(* Logix 5000 project; controller cal1632 1756-L62 rev 16.20; software revision 16.05; part 8 of 57 *)
(* tags used below, declared in another part *)
   FAULT : BOOL;
   p01_r15_footage_ft : REAL;
   p01_real_to_hmi : REAL[112];
   p01r09_pb_global_reset : BOOL;
   p02_real_to_hmi : hmi_real;
   p02r06 : routine;
   p02r06_timer_fault : TIMER[4];
   p02r06_timer_warning : TIMER[4];
   p02r07 : routine;
   p02r07_timer_fault : TIMER[4];
   p02r07_timer_warning : TIMER[4];
   p02r08 : routine;
   p02r08_timer_fault : TIMER[4];
   p02r08_timer_warning : TIMER[4];
   p02r09 : routine;
   p02r09_timer_fault : TIMER[4];
   p02r09_timer_warning : TIMER[4];
   p02r10 : routine;
   p02r10_timer_fault : TIMER[4];
   p02r10_timer_warning : TIMER[4];
   p02r11 : routine;
   p02r11_timer_fault : TIMER[4];
   p02r11_timer_warning : TIMER[4];
   p11_real_to_hmi : REAL[112];
   p12_real_to_hmi : REAL[112];
   p13_real_to_hmi : REAL[112];
   p19_real_to_hmi : REAL[80];
   p20_real_to_hmi : REAL[112];
   p21_real_to_hmi : REAL[112];
   p22_real_to_hmi : REAL[112];
   p23_real_to_hmi : REAL[112];
   p24_real_to_hmi : REAL[112];
   p25_real_to_hmi : REAL[112];
   p26_real_to_hmi : REAL[112];
   p27_real_to_hmi : REAL[112];
   p28_real_to_hmi : REAL[112];
   p29_real_to_hmi : REAL[112];
(* P02_MOP_HMI_Iface, continued *)

ROUTINE R06_Real_to_HMI   (* ladder *)
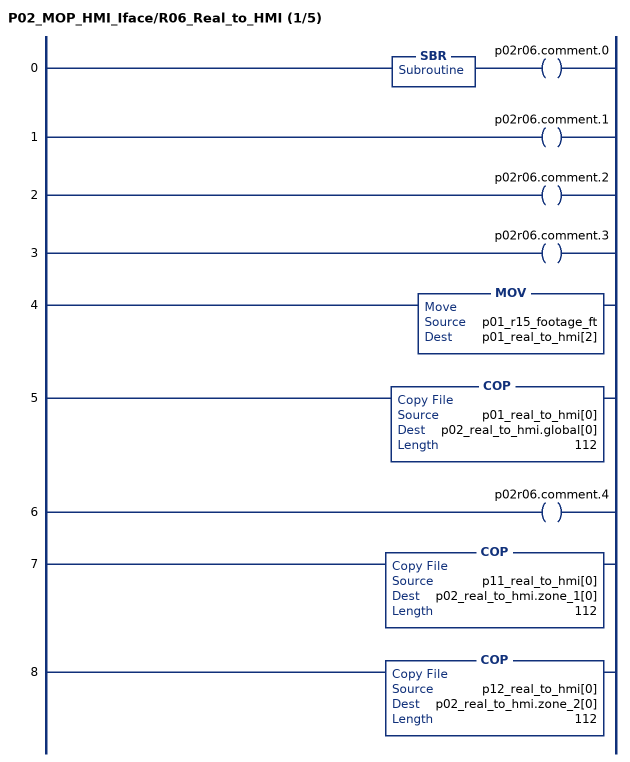
   0: SBR()OTE(p02r06.comment.0);
   1: OTE(p02r06.comment.1);
   2: OTE(p02r06.comment.2);
   3: OTE(p02r06.comment.3);
   4: MOV(p01_r15_footage_ft,p01_real_to_hmi[2]);
   5: COP(p01_real_to_hmi[0],p02_real_to_hmi.global[0],112);
   6: OTE(p02r06.comment.4);
   7: COP(p11_real_to_hmi[0],p02_real_to_hmi.zone_1[0],112);
   8: COP(p12_real_to_hmi[0],p02_real_to_hmi.zone_2[0],112);
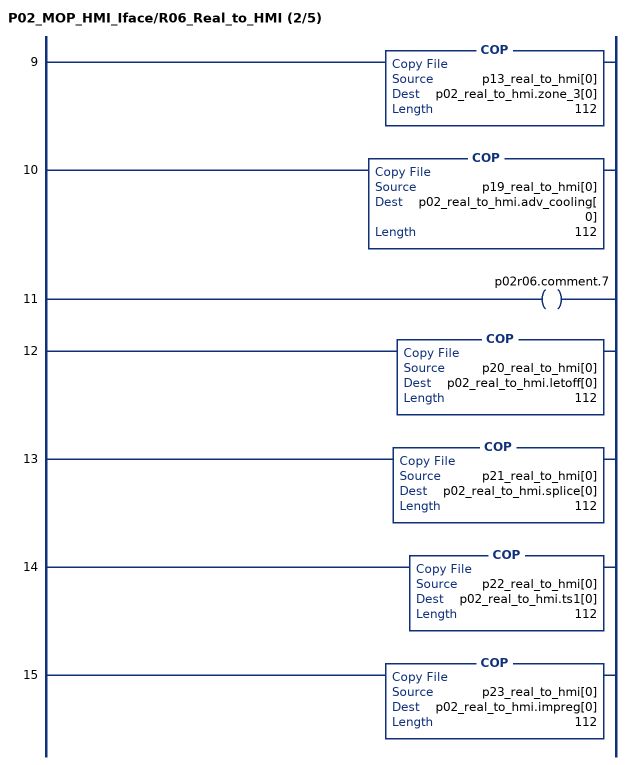
   9: COP(p13_real_to_hmi[0],p02_real_to_hmi.zone_3[0],112);
   10: COP(p19_real_to_hmi[0],p02_real_to_hmi.adv_cooling[0],112);
   11: OTE(p02r06.comment.7);
   12: COP(p20_real_to_hmi[0],p02_real_to_hmi.letoff[0],112);
   13: COP(p21_real_to_hmi[0],p02_real_to_hmi.splice[0],112);
   14: COP(p22_real_to_hmi[0],p02_real_to_hmi.ts1[0],112);
   15: COP(p23_real_to_hmi[0],p02_real_to_hmi.impreg[0],112);
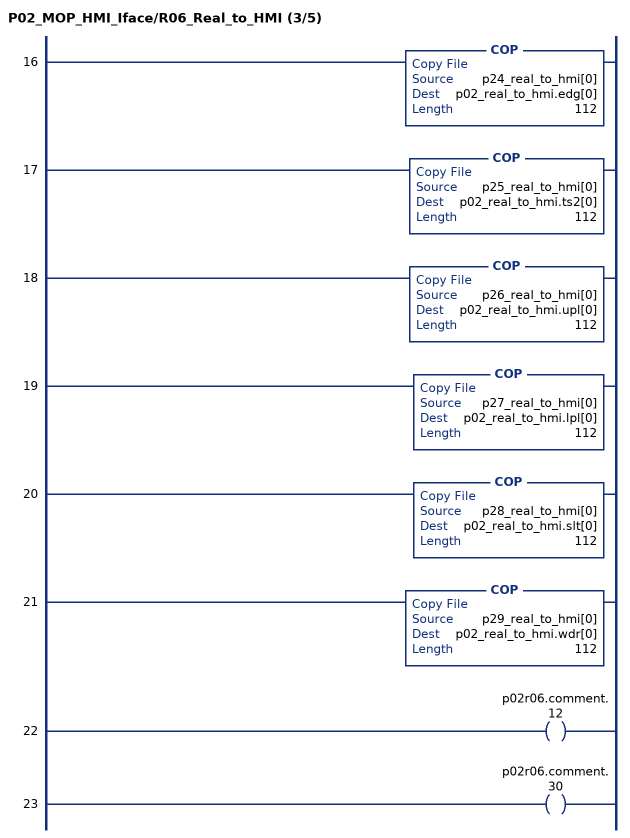
   16: COP(p24_real_to_hmi[0],p02_real_to_hmi.edg[0],112);
   17: COP(p25_real_to_hmi[0],p02_real_to_hmi.ts2[0],112);
   18: COP(p26_real_to_hmi[0],p02_real_to_hmi.upl[0],112);
   19: COP(p27_real_to_hmi[0],p02_real_to_hmi.lpl[0],112);
   20: COP(p28_real_to_hmi[0],p02_real_to_hmi.slt[0],112);
   21: COP(p29_real_to_hmi[0],p02_real_to_hmi.wdr[0],112);
   22: OTE(p02r06.comment.12);
   23: OTE(p02r06.comment.30);
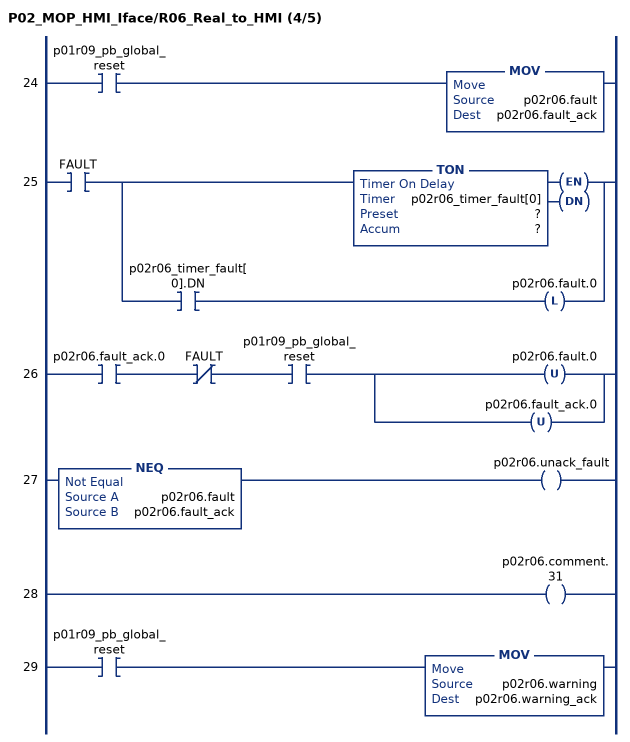
   24: XIC(p01r09_pb_global_reset)MOV(p02r06.fault,p02r06.fault_ack);
   25: XIC(FAULT)[TON(p02r06_timer_fault[0],?,?) ,XIC(p02r06_timer_fault[0].DN) OTL(p02r06.fault.0) ];
   26: XIC(p02r06.fault_ack.0)XIO(FAULT)XIC(p01r09_pb_global_reset)[OTU(p02r06.fault.0) ,OTU(p02r06.fault_ack.0) ];
   27: NEQ(p02r06.fault,p02r06.fault_ack)OTE(p02r06.unack_fault);
   28: OTE(p02r06.comment.31);
   29: XIC(p01r09_pb_global_reset)MOV(p02r06.warning,p02r06.warning_ack);
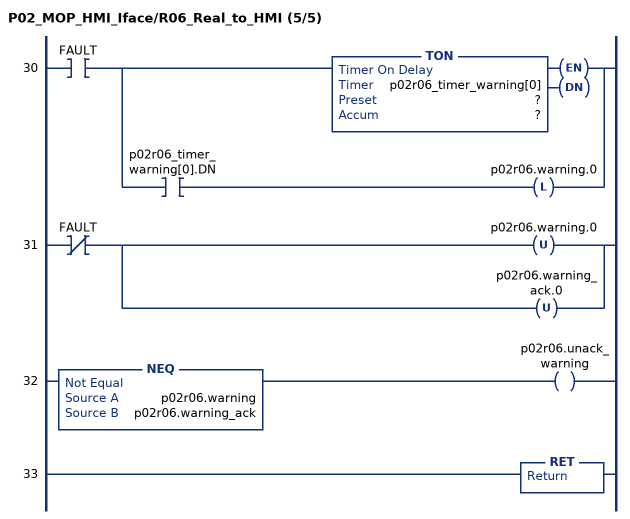
   30: XIC(FAULT)[TON(p02r06_timer_warning[0],?,?) ,XIC(p02r06_timer_warning[0].DN) OTL(p02r06.warning.0) ];
   31: XIO(FAULT)[OTU(p02r06.warning.0) ,OTU(p02r06.warning_ack.0) ];
   32: NEQ(p02r06.warning,p02r06.warning_ack)OTE(p02r06.unack_warning);
   33: RET();
END_ROUTINE

ROUTINE R07_Alarms   (* ladder *)
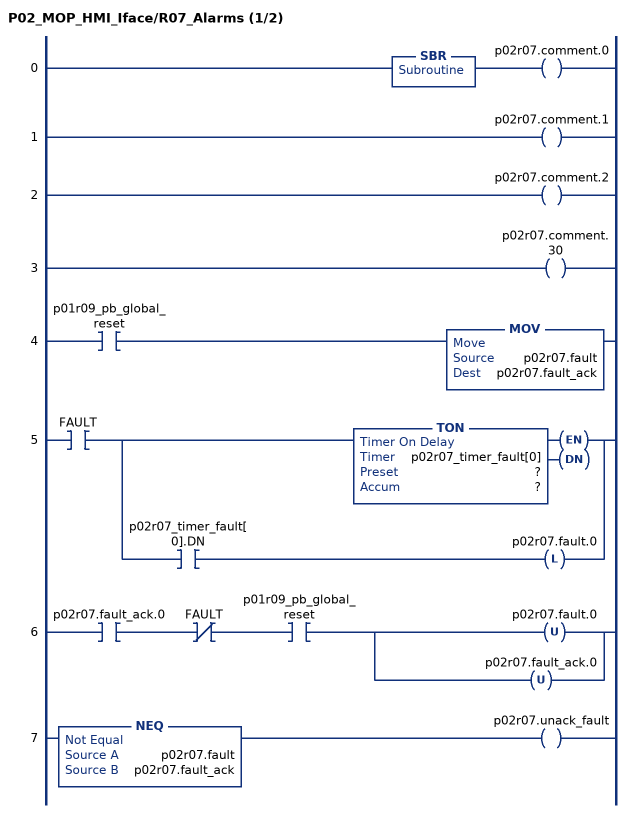
   0: SBR()OTE(p02r07.comment.0);
   1: OTE(p02r07.comment.1);
   2: OTE(p02r07.comment.2);
   3: OTE(p02r07.comment.30);
   4: XIC(p01r09_pb_global_reset)MOV(p02r07.fault,p02r07.fault_ack);
   5: XIC(FAULT)[TON(p02r07_timer_fault[0],?,?) ,XIC(p02r07_timer_fault[0].DN) OTL(p02r07.fault.0) ];
   6: XIC(p02r07.fault_ack.0)XIO(FAULT)XIC(p01r09_pb_global_reset)[OTU(p02r07.fault.0) ,OTU(p02r07.fault_ack.0) ];
   7: NEQ(p02r07.fault,p02r07.fault_ack)OTE(p02r07.unack_fault);
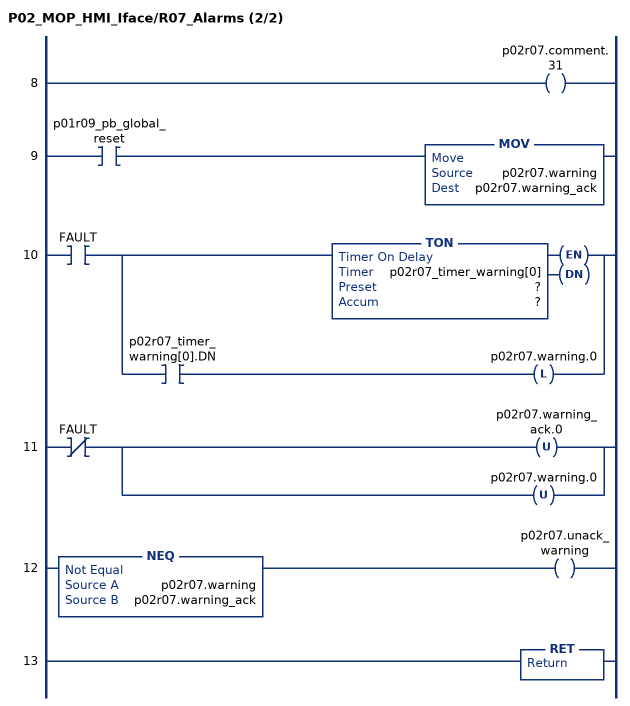
   8: OTE(p02r07.comment.31);
   9: XIC(p01r09_pb_global_reset)MOV(p02r07.warning,p02r07.warning_ack);
   10: XIC(FAULT)[TON(p02r07_timer_warning[0],?,?) ,XIC(p02r07_timer_warning[0].DN) OTL(p02r07.warning.0) ];
   11: XIO(FAULT)[OTU(p02r07.warning_ack.0) ,OTU(p02r07.warning.0) ];
   12: NEQ(p02r07.warning,p02r07.warning_ack)OTE(p02r07.unack_warning);
   13: RET();
END_ROUTINE

ROUTINE R08_Warnings   (* ladder *)
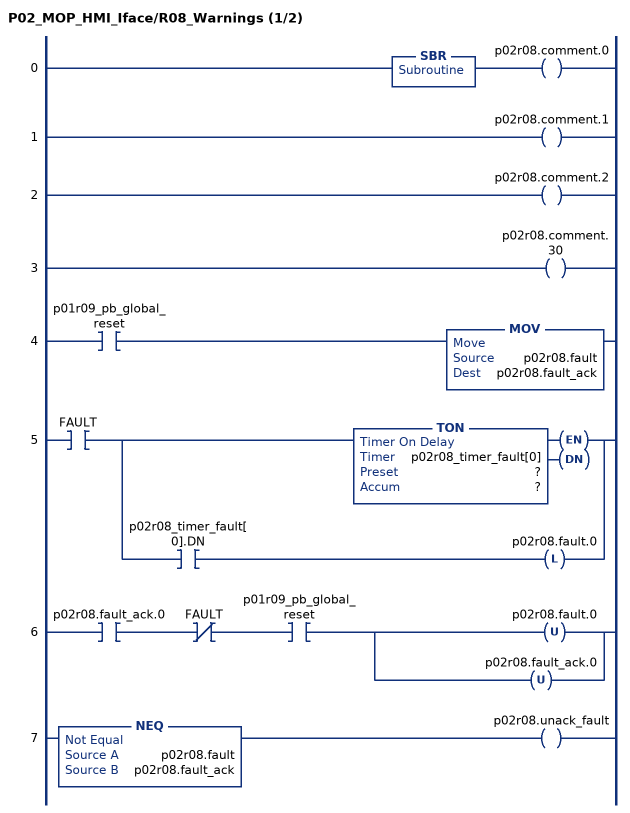
   0: SBR()OTE(p02r08.comment.0);
   1: OTE(p02r08.comment.1);
   2: OTE(p02r08.comment.2);
   3: OTE(p02r08.comment.30);
   4: XIC(p01r09_pb_global_reset)MOV(p02r08.fault,p02r08.fault_ack);
   5: XIC(FAULT)[TON(p02r08_timer_fault[0],?,?) ,XIC(p02r08_timer_fault[0].DN) OTL(p02r08.fault.0) ];
   6: XIC(p02r08.fault_ack.0)XIO(FAULT)XIC(p01r09_pb_global_reset)[OTU(p02r08.fault.0) ,OTU(p02r08.fault_ack.0) ];
   7: NEQ(p02r08.fault,p02r08.fault_ack)OTE(p02r08.unack_fault);
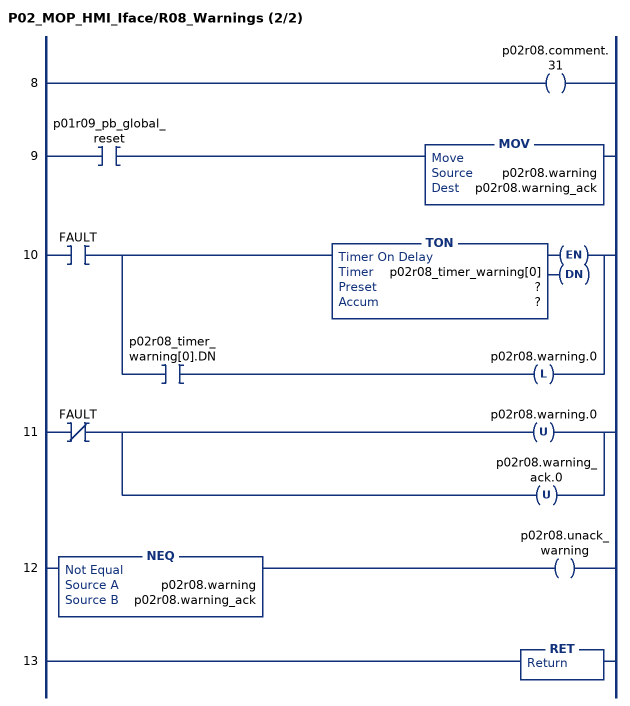
   8: OTE(p02r08.comment.31);
   9: XIC(p01r09_pb_global_reset)MOV(p02r08.warning,p02r08.warning_ack);
   10: XIC(FAULT)[TON(p02r08_timer_warning[0],?,?) ,XIC(p02r08_timer_warning[0].DN) OTL(p02r08.warning.0) ];
   11: XIO(FAULT)[OTU(p02r08.warning.0) ,OTU(p02r08.warning_ack.0) ];
   12: NEQ(p02r08.warning,p02r08.warning_ack)OTE(p02r08.unack_warning);
   13: RET();
END_ROUTINE

ROUTINE R09_Maintenance   (* ladder *)
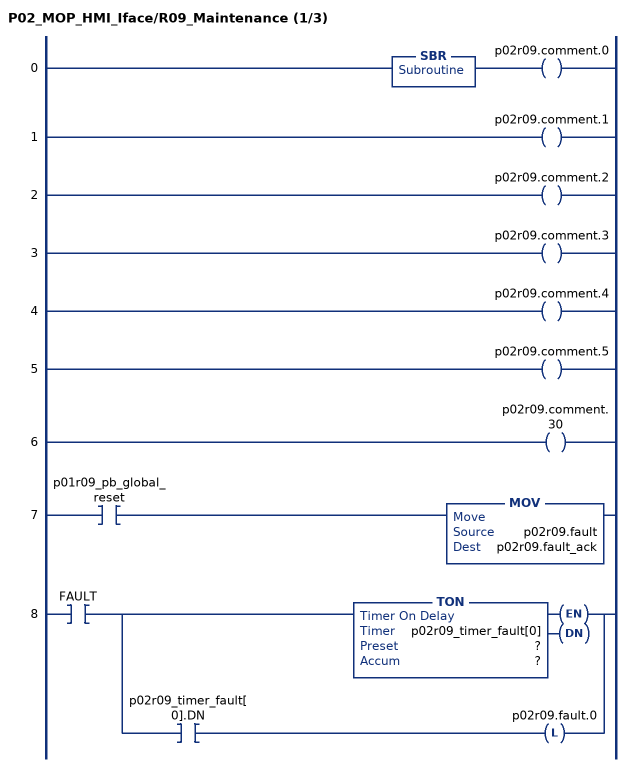
   0: SBR()OTE(p02r09.comment.0);
   1: OTE(p02r09.comment.1);
   2: OTE(p02r09.comment.2);
   3: OTE(p02r09.comment.3);
   4: OTE(p02r09.comment.4);
   5: OTE(p02r09.comment.5);
   6: OTE(p02r09.comment.30);
   7: XIC(p01r09_pb_global_reset)MOV(p02r09.fault,p02r09.fault_ack);
   8: XIC(FAULT)[TON(p02r09_timer_fault[0],?,?) ,XIC(p02r09_timer_fault[0].DN) OTL(p02r09.fault.0) ];
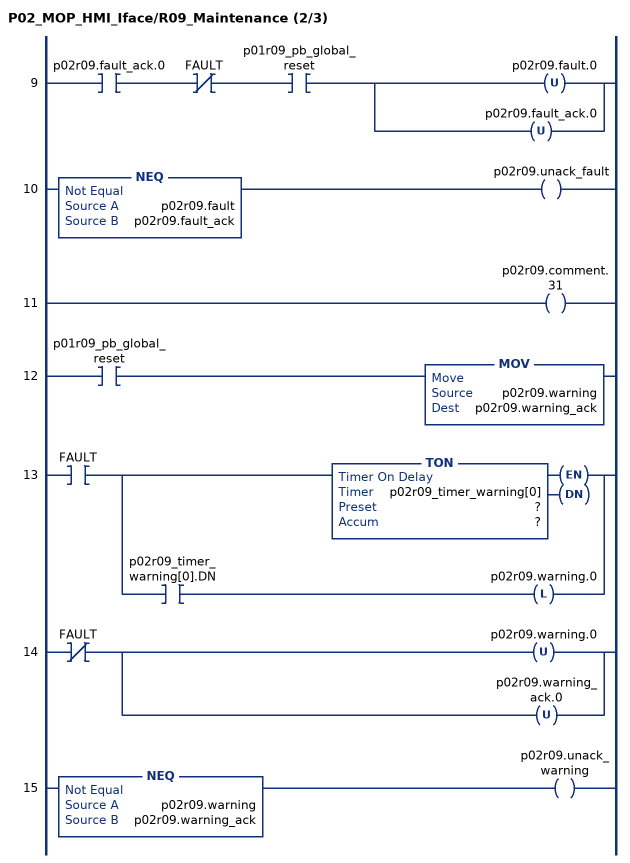
   9: XIC(p02r09.fault_ack.0)XIO(FAULT)XIC(p01r09_pb_global_reset)[OTU(p02r09.fault.0) ,OTU(p02r09.fault_ack.0) ];
   10: NEQ(p02r09.fault,p02r09.fault_ack)OTE(p02r09.unack_fault);
   11: OTE(p02r09.comment.31);
   12: XIC(p01r09_pb_global_reset)MOV(p02r09.warning,p02r09.warning_ack);
   13: XIC(FAULT)[TON(p02r09_timer_warning[0],?,?) ,XIC(p02r09_timer_warning[0].DN) OTL(p02r09.warning.0) ];
   14: XIO(FAULT)[OTU(p02r09.warning.0) ,OTU(p02r09.warning_ack.0) ];
   15: NEQ(p02r09.warning,p02r09.warning_ack)OTE(p02r09.unack_warning);
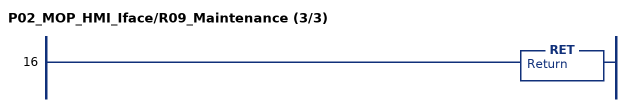
   16: RET();
END_ROUTINE

ROUTINE R10   (* ladder *)
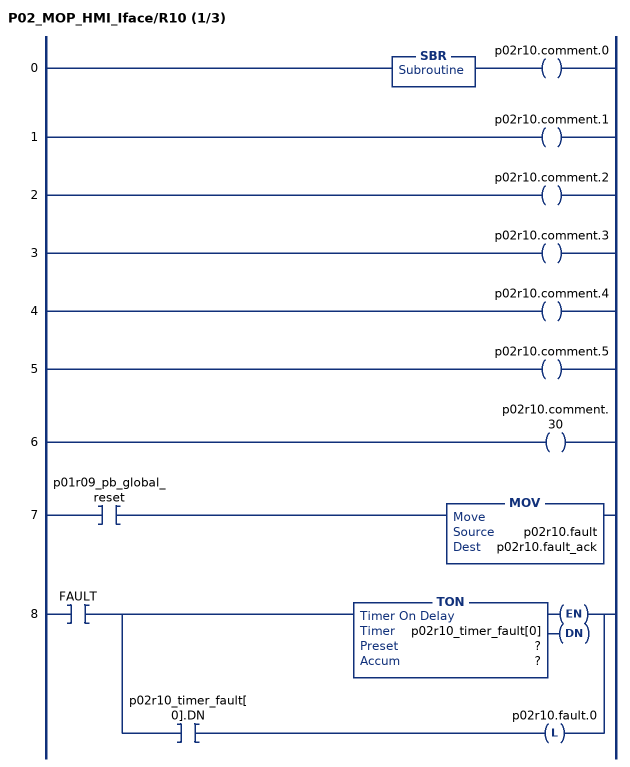
   0: SBR()OTE(p02r10.comment.0);
   1: OTE(p02r10.comment.1);
   2: OTE(p02r10.comment.2);
   3: OTE(p02r10.comment.3);
   4: OTE(p02r10.comment.4);
   5: OTE(p02r10.comment.5);
   6: OTE(p02r10.comment.30);
   7: XIC(p01r09_pb_global_reset)MOV(p02r10.fault,p02r10.fault_ack);
   8: XIC(FAULT)[TON(p02r10_timer_fault[0],?,?) ,XIC(p02r10_timer_fault[0].DN) OTL(p02r10.fault.0) ];
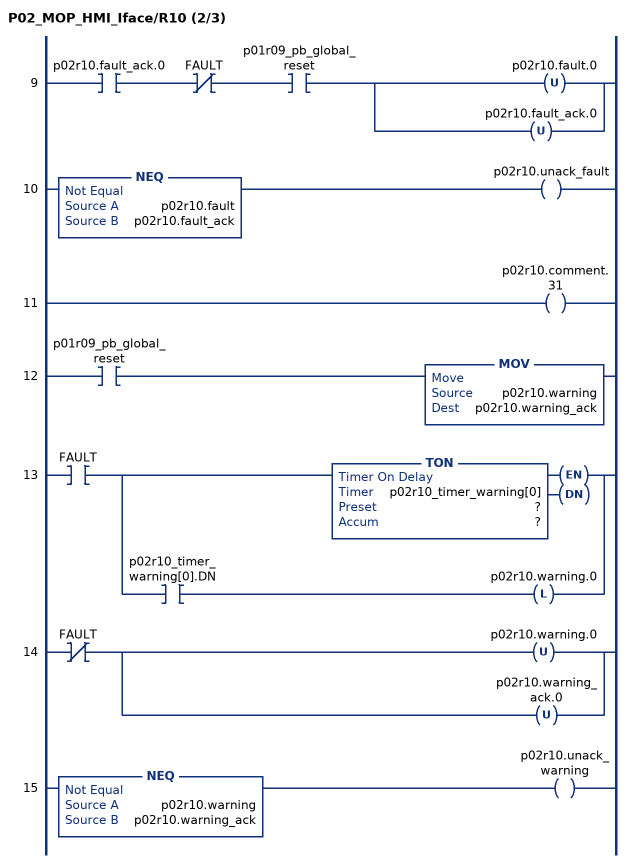
   9: XIC(p02r10.fault_ack.0)XIO(FAULT)XIC(p01r09_pb_global_reset)[OTU(p02r10.fault.0) ,OTU(p02r10.fault_ack.0) ];
   10: NEQ(p02r10.fault,p02r10.fault_ack)OTE(p02r10.unack_fault);
   11: OTE(p02r10.comment.31);
   12: XIC(p01r09_pb_global_reset)MOV(p02r10.warning,p02r10.warning_ack);
   13: XIC(FAULT)[TON(p02r10_timer_warning[0],?,?) ,XIC(p02r10_timer_warning[0].DN) OTL(p02r10.warning.0) ];
   14: XIO(FAULT)[OTU(p02r10.warning.0) ,OTU(p02r10.warning_ack.0) ];
   15: NEQ(p02r10.warning,p02r10.warning_ack)OTE(p02r10.unack_warning);
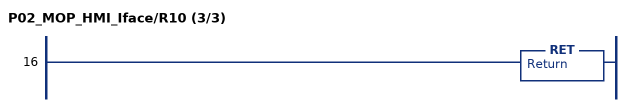
   16: RET();
END_ROUTINE

ROUTINE R11   (* ladder *)
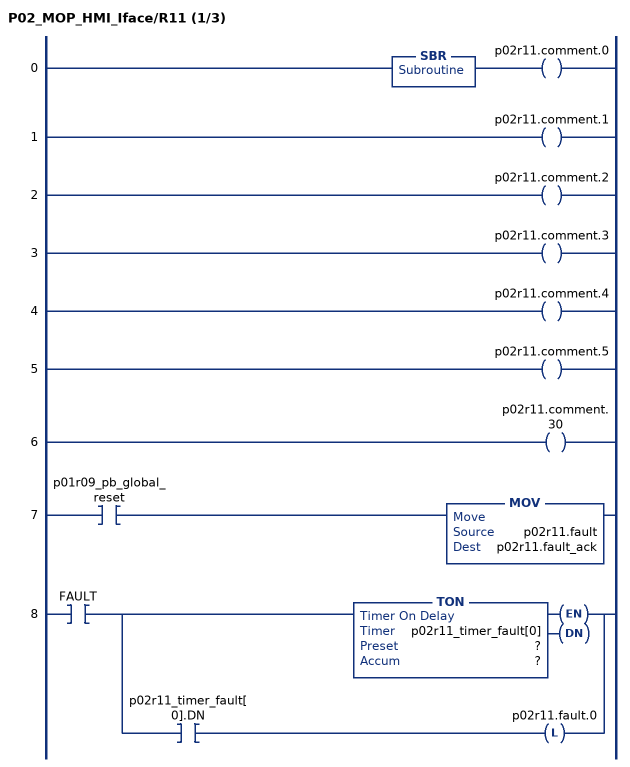
   0: SBR()OTE(p02r11.comment.0);
   1: OTE(p02r11.comment.1);
   2: OTE(p02r11.comment.2);
   3: OTE(p02r11.comment.3);
   4: OTE(p02r11.comment.4);
   5: OTE(p02r11.comment.5);
   6: OTE(p02r11.comment.30);
   7: XIC(p01r09_pb_global_reset)MOV(p02r11.fault,p02r11.fault_ack);
   8: XIC(FAULT)[TON(p02r11_timer_fault[0],?,?) ,XIC(p02r11_timer_fault[0].DN) OTL(p02r11.fault.0) ];
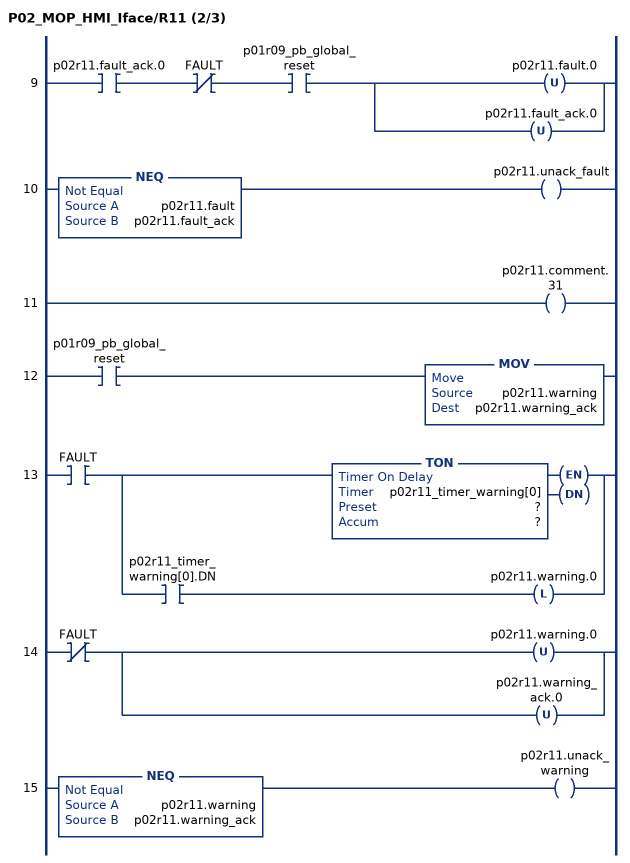
   9: XIC(p02r11.fault_ack.0)XIO(FAULT)XIC(p01r09_pb_global_reset)[OTU(p02r11.fault.0) ,OTU(p02r11.fault_ack.0) ];
   10: NEQ(p02r11.fault,p02r11.fault_ack)OTE(p02r11.unack_fault);
   11: OTE(p02r11.comment.31);
   12: XIC(p01r09_pb_global_reset)MOV(p02r11.warning,p02r11.warning_ack);
   13: XIC(FAULT)[TON(p02r11_timer_warning[0],?,?) ,XIC(p02r11_timer_warning[0].DN) OTL(p02r11.warning.0) ];
   14: XIO(FAULT)[OTU(p02r11.warning.0) ,OTU(p02r11.warning_ack.0) ];
   15: NEQ(p02r11.warning,p02r11.warning_ack)OTE(p02r11.unack_warning);
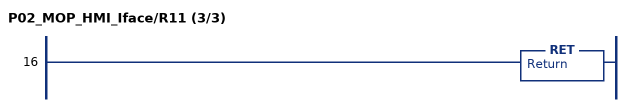
   16: RET();
END_ROUTINE
